KUKA KRL program: style1app1opt1.src, style1app1opt1.dat

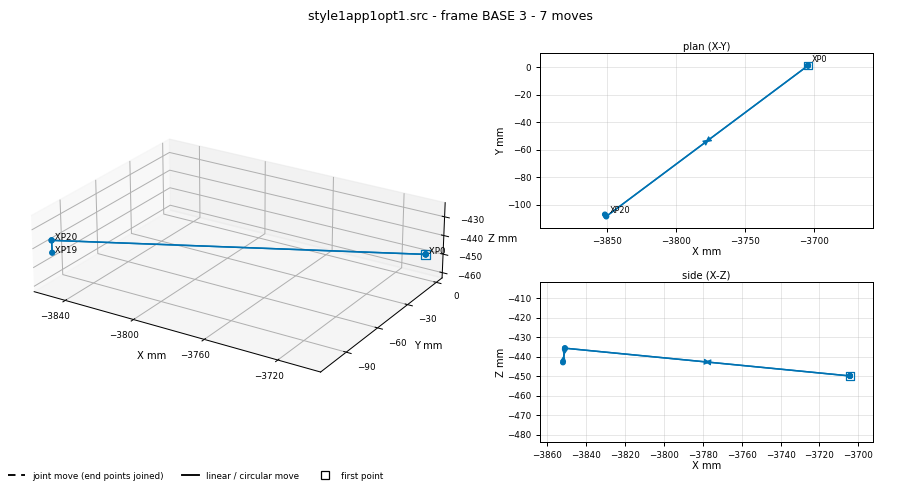
[picture p0: tool path of style1app1opt1.src in frame BASE 3, 7 of 7 moves have a stored position in this frame; points joined in program order, loops and branches not executed]
--- style1app1opt1.src ---
&ACCESS RVO1
&REL 339
&COMMENT 03-10-R1 PNW1 NUT 1
&PARAM EDITMASK = *
&PARAM TEMPLATE = C:\KRC\TP\Nutweld\Template\NutWeld_Vorgabe
&PARAM DISKPATH = KRC:\R1\Program\StyleApps\Options
DEF style1app1opt1( )
   ;FOLD INI
      ;FOLD BASISTECH INI
         GLOBAL INTERRUPT DECL 3 WHEN $STOPMESS==TRUE DO IR_STOPM ( )
         INTERRUPT ON 3
         BAS (#INITMOV,0 )
      ;ENDFOLD (BASISTECH INI)
      ;FOLD NutWeld
      ;ENDFOLD (NutWeld)
      ;FOLD USER INI
         ;Make your modifications here

      ;ENDFOLD (USER INI)
   ;ENDFOLD (INI)
;********************************
; Gestamp Standards
; Line - BMW G65 (cell 03)
; Robot 03-10-R1 (BMW-03-10-R1-PNW1)
; Application - WELD NUT 1 (PN1) AT THE CENTERLINE PEDESTAL
;********************************
; CALLED BY Style1Opt1. APPROACH THE PEDESTAL (BASE 3 "NUT WELDER"), WAIT FOR THE NUT PRELOAD
; (NUT_READY), MOVE THE PART TO THE WELD POSITION P19, WELD WITH CENTERLINE_WELD (NOT IN DRY
; CYCLE), LEAVE THE PEDESTAL.
;WARNING: BEFORE THE ROBOT MOVES IN, ONLY NUT_READY IS CHECKED - NOT GUN OPEN, CLAMP OPEN OR
;  QFP RETURNED (F01)
;NOTE: THE PEDESTAL MOVES MIX BASE MODE AND EXTERNAL-TCP MODE (extTCP); THE WELD POSITION
;  P19 IS TAUGHT IN BASE MODE (F22)

;APPROACH THE PEDESTAL - P0, P8
;FOLD PTP P0 CONT Vel=100 % PDAT0 Tool[1]:TOOL 1 Base[3]:NUT WELDER extTCP;%{PE}%R 8.3.43,%MKUKATPBASIS,%CMOVE,%VPTP,%P 1:PTP, 2:P0, 3:C_DIS, 5:100, 7:PDAT0
$BWDSTART=FALSE
PDAT_ACT=PPDAT0
FDAT_ACT=FP0
BAS(#PTP_PARAMS,100)
PTP XP0 C_DIS
;ENDFOLD
;FOLD LIN P8 CONT Vel=2 m/s CPDAT12 Tool[1]:TOOL 1 Base[3]:NUT WELDER extTCP;%{PE}%R 8.3.43,%MKUKATPBASIS,%CMOVE,%VLIN,%P 1:LIN, 2:P8, 3:C_DIS C_DIS, 5:2, 7:CPDAT12
$BWDSTART=FALSE
LDAT_ACT=LCPDAT12
FDAT_ACT=FP8
BAS(#CP_PARAMS,2)
LIN XP8 C_DIS C_DIS
;ENDFOLD
;NOTE: RETRY_NUT1 IS THE TARGET OF THE NUT_WELD_RETRY BRANCH BELOW, WHICH NEVER RUNS (F24)
RETRY_NUT1:
;WAIT NUT PRELOADED - NUT_READY (SET BY PRELOAD WHEN THE NUT IS ON THE LOWER PIN)
;NOTE: NO TIMEOUT, NO MESSAGE (F15). IN DRY CYCLE NOTHING SETS IT: THE CYCLE HANGS HERE (F04)
;NOTE: NUT_READY IS NOT CLEARED AFTER A WELD: IF THE PICK TRIGGER WAS SKIPPED, THE TRUE OF THE
;  LAST CYCLE LETS THE ROBOT IN WITH NO NUT FED (F14)
WAIT FOR NUT_READY== TRUE

;MOVE IN - P20 (2 M/S), THEN THE WELD POSITION P19 OUTSIDE DRY CYCLE
;FOLD LIN P20 CONT Vel=2 m/s CPDAT8 Tool[1]:TOOL 1 Base[3]:NUT WELDER;%{PE}%R 8.3.43,%MKUKATPBASIS,%CMOVE,%VLIN,%P 1:LIN, 2:P20, 3:C_DIS C_DIS, 5:2, 7:CPDAT8
$BWDSTART=FALSE
LDAT_ACT=LCPDAT8
FDAT_ACT=FP20
BAS(#CP_PARAMS,2)
LIN XP20 C_DIS C_DIS
;ENDFOLD

;DRY CYCLE (SIGNAL $IN[4] di004UseDryCycle ON): NO WELD POSITION, NO WELD - JUMP TO DRY1 (F05)
IF di004UseDryCycle==TRUE THEN

GOTO DRY1
ELSE

;FOLD LIN P19 Vel=2 m/s CPDAT18 Tool[1]:TOOL 1 Base[3]:NUT WELDER;%{PE}%R 8.3.43,%MKUKATPBASIS,%CMOVE,%VLIN,%P 1:LIN, 2:P19, 3:, 5:2, 7:CPDAT18
$BWDSTART=FALSE
LDAT_ACT=LCPDAT18
FDAT_ACT=FP19
BAS(#CP_PARAMS,2)
LIN XP19
;ENDFOLD
;NUT WELD AT THE PEDESTAL (CENTERLINE_WELD: CLAMP, GUN, INTENSIFY, BOSCH WELD, GUN OPEN)
CENTERLINE_WELD()

ENDIF
DRY1:
;LEAVE THE PEDESTAL - P20, P8, P0

;FOLD LIN P20 CONT Vel=2 m/s CPDAT16 Tool[1]:TOOL 1 Base[3]:NUT WELDER;%{PE}%R 8.3.43,%MKUKATPBASIS,%CMOVE,%VLIN,%P 1:LIN, 2:P20, 3:C_DIS C_DIS, 5:2, 7:CPDAT16
$BWDSTART=FALSE
LDAT_ACT=LCPDAT16
FDAT_ACT=FP20
BAS(#CP_PARAMS,2)
LIN XP20 C_DIS C_DIS
;ENDFOLD


;NOTE: NUT_WELD_RETRY IS NEVER SET TRUE - THIS RETRY BRANCH IS DEAD CODE (F24, GESTAMP POINT 17)
IF NUT_WELD_RETRY THEN
   NUT_WELD_RETRY=FALSE

   GOTO RETRY_NUT1
ENDIF

;FOLD LIN P8 CONT Vel=2 m/s CPDAT17 Tool[1]:TOOL 1 Base[3]:NUT WELDER extTCP;%{PE}%R 8.3.43,%MKUKATPBASIS,%CMOVE,%VLIN,%P 1:LIN, 2:P8, 3:C_DIS C_DIS, 5:2, 7:CPDAT17
$BWDSTART=FALSE
LDAT_ACT=LCPDAT17
FDAT_ACT=FP8
BAS(#CP_PARAMS,2)
LIN XP8 C_DIS C_DIS
;ENDFOLD
;NEXT NUT - TRIGGER IN THE P0 FOLD (DISTANCE = 0: FIRES WHEN THE MOTION STARTS, PRIO -1):
;Request_next_nut() CLEARS NEXT_NUT_READY AND STARTS THE PRELOAD OF NUT 2 (NUT_STAR=TRUE)
;WARNING: THE TRIGGER WAS TYPED BY HAND INSIDE THE INLINE FORM: A TOUCH UP OF P0 DELETES IT
;  AND NUT 2 WAITS FOREVER FOR NEXT_NUT_READY (F32, GESTAMP POINT 20)
;FOLD PTP P0 Vel=100 % PDAT18 Tool[1]:TOOL 1 Base[3]:NUT WELDER extTCP;%{PE}%R 8.3.43,%MKUKATPBASIS,%CMOVE,%VPTP,%P 1:PTP, 2:P0, 3:, 5:100, 7:PDAT18
$BWDSTART=FALSE
PDAT_ACT=PPDAT18
FDAT_ACT=FP0
BAS(#PTP_PARAMS,100)
TRIGGER WHEN DISTANCE = 0 DELAY = 0 DO Request_next_nut() PRIO= -1
PTP XP0
;ENDFOLD
END

--- style1app1opt1.dat ---
&ACCESS RVO1
&REL 339
&COMMENT NUT1
&PARAM EDITMASK = *
&PARAM TEMPLATE = C:\KRC\TP\Nutweld\Template\NutWeld_Vorgabe
&PARAM DISKPATH = KRC:\R1\Program\StyleApps\Options
DEFDAT  style1app1opt1
;FOLD EXTERNAL DECLARATIONS;%{PE}%MKUKATPBASIS,%CEXT,%VCOMMON,%P
;FOLD BASISTECH EXT;%{PE}%MKUKATPBASIS,%CEXT,%VEXT,%P
EXT  BAS (BAS_COMMAND  :IN,REAL  :IN )
;ENDFOLD (BASISTECH EXT)
;FOLD NutWeld
;ENDFOLD (NutWeld)
;FOLD USER EXT;%{E}%MKUKATPUSER,%CEXT,%VEXT,%P
;Make here your modifications
;ENDFOLD (USER EXT)
DECL E6POS XP20={X -3850.82104,Y -108.397034,Z -435.544800,A -178.432037,B 0.654220462,C -179.967712,S 2,T 34,E1 0.0,E2 0.0,E3 0.0,E4 0.0,E5 0.0,E6 0.0}
DECL FDAT FP20={TOOL_NO 1,BASE_NO 3,IPO_FRAME #BASE,POINT2[] " ",TQ_STATE FALSE}
;ENDFOLD (EXTERNAL DECLARATIONS)








DECL FDAT FPNW1={TOOL_NO 2,BASE_NO 1,IPO_FRAME #TCP,POINT2[] " ",TQ_STATE FALSE}
DECL E6POS XPNW1={X 123.774101,Y 312.995331,Z -88.6478,A 8.71582699,B 8.82717705,C 1.11576855,S 2,T 3,E1 0.0,E2 0.0,E3 0.0,E4 0.0,E5 0.0,E6 0.0}
DECL NutWeld_SUGG_T LAST_NutWeld={POINT1[] "PNW1_SPOT7              ",POINT2[] "PNW0                    ",CP_PARAMS[] "CPDATNutWeld0           ",PTP_PARAMS[] "PDATNutWeld0            ",CONT[] "C_PTP                   ",CP_VEL[] "2                       ",PTP_VEL[] "100                     ",SYNC_PARAMS[] "SYNCDAT                 ",SPL_NAME[] "S0                      ",NutWeld_PARAMS[] "NutData1_7              ",GunNr 1,SpotNr 7,Offset 45}
DECL BASIS_SUGG_T LAST_BASIS={POINT1[] "P0                      ",POINT2[] "P0                      ",CP_PARAMS[] "CPDAT0                  ",PTP_PARAMS[] "PDAT0                   ",CONT[] "                        ",CP_VEL[] "2                       ",PTP_VEL[] " 100                    ",SYNC_PARAMS[] "SYNCDAT                 ",SPL_NAME[] "S0                      ",A_PARAMS[] "ADAT0                   "}
DECL PDAT PPDAT0={VEL 100.000,ACC 100.000,APO_DIST 100.000,APO_MODE #CDIS,GEAR_JERK 50.0000,EXAX_IGN 0}
DECL E6POS XP0={X -3704.29346,Y 1.10223198,Z -449.805786,A -178.368118,B 0.266879767,C 179.968445,S 2,T 34,E1 0.0,E2 0.0,E3 0.0,E4 0.0,E5 0.0,E6 0.0}
DECL FDAT FP0={TOOL_NO 1,BASE_NO 3,IPO_FRAME #TCP,POINT2[] " ",TQ_STATE FALSE}
DECL MODULEPARAM_T LAST_TP_PARAMS={PARAMS[] "NutWeld_CmdPos=Weld; NutWeld_Move=LIN; NutWeld_NutWeldDat=NutData1_7; NutWeld_NWGunNr=1; NutWeld_NWSpotNr=7; NutWeld_NWOffset=45; Kuka.MoveDataName=gAboveWeld; Kuka.VelocityPath=2; Kuka.PointName=PNW1_CNTRH_SPOT7; Kuka.BlendingEnabled=False; Kuka.FrameData.tq_state=False; Kuka.FrameData.base_no=1; Kuka.FrameData.tool_no=1; Kuka.FrameData.ipo_frame=#TCP; Kuka.FrameData.point2=; Kuka.MovementData.apo_fac=50; Kuka.MovementData.apo_dist=100; Kuka.MovementData.axis_acc=100; Kuka.MovementData.axis_vel=100; Kuka.MovementData.circ_typ=#BASE; Kuka.MovementData.exax_ign=0; Kuka.MovementData.jerk_fac=50; Kuka.MovementData.ori_typ=#VAR; Kuka.MovementData.acc=100; Kuka.MovementData.gear_jerk=50  "}
DECL E6POS XP8={X -3704.29346,Y 1.10223198,Z -449.805786,A -178.368118,B 0.266879767,C 179.968445,S 2,T 34,E1 0.0,E2 0.0,E3 0.0,E4 0.0,E5 0.0,E6 0.0}
DECL FDAT FP8={TOOL_NO 1,BASE_NO 3,IPO_FRAME #TCP,POINT2[] " ",TQ_STATE FALSE}
DECL LDAT LCPDAT8={VEL 2.00000,ACC 100.000,APO_DIST 100.000,APO_FAC 50.0000,AXIS_VEL 100.000,AXIS_ACC 100.000,ORI_TYP #VAR,CIRC_TYP #BASE,JERK_FAC 50.0000,GEAR_JERK 50.0000,EXAX_IGN 0}
DECL LDAT LCPDAT12={VEL 2.00000,ACC 100.000,APO_DIST 100.000,APO_FAC 50.0000,AXIS_VEL 100.000,AXIS_ACC 100.000,ORI_TYP #VAR,CIRC_TYP #BASE,JERK_FAC 50.0000,GEAR_JERK 50.0000,EXAX_IGN 0}
DECL LDAT LCPDAT16={VEL 2.00000,ACC 100.000,APO_DIST 100.000,APO_FAC 50.0000,AXIS_VEL 100.000,AXIS_ACC 100.000,ORI_TYP #VAR,CIRC_TYP #BASE,JERK_FAC 50.0000,GEAR_JERK 50.0000,EXAX_IGN 0}
DECL LDAT LCPDAT17={VEL 2.00000,ACC 100.000,APO_DIST 100.000,APO_FAC 50.0000,AXIS_VEL 100.000,AXIS_ACC 100.000,ORI_TYP #VAR,CIRC_TYP #BASE,JERK_FAC 50.0000,GEAR_JERK 50.0000,EXAX_IGN 0}
DECL PDAT PPDAT18={VEL 100.000,ACC 100.000,APO_DIST 100.000,APO_MODE #CDIS,GEAR_JERK 50.0000,EXAX_IGN 0}
DECL E6POS XP19={X -3851.81445,Y -107.010963,Z -442.857483,A -178.432037,B 0.654220223,C -179.967712,S 2,T 34,E1 0.0,E2 0.0,E3 0.0,E4 0.0,E5 0.0,E6 0.0}
DECL FDAT FP19={TOOL_NO 1,BASE_NO 3,IPO_FRAME #BASE,POINT2[] " ",TQ_STATE FALSE}
DECL LDAT LCPDAT18={VEL 2.00000,ACC 100.000,APO_DIST 100.000,APO_FAC 50.0000,AXIS_VEL 100.000,AXIS_ACC 100.000,ORI_TYP #VAR,CIRC_TYP #BASE,JERK_FAC 50.0000,GEAR_JERK 50.0000,EXAX_IGN 0}
ENDDAT
